FUNCTION IsOk : BOOL
VAR_INPUT
	eResult			: Result;
END_VAR
VAR_OUTPUT
	eCarry			: Result;
END_VAR

IsOk := eResult > 0;
eCarry := eResult;

END_FUNCTION

(* stored: Version 1.1.0.1
   POU IsOk: Id {d5d94619-7758-428d-8e9e-49647c79f7a4}, SpecialFunc None *)
